SUBAPPLICATION Uebung_012d_AR (* Numeric Value Input PHYS und Speichern NVS (AR Adapter, plain) *)
  (* Standard: 61499-2; Description: Copyright (c) 2026 Meisterschulen am Ostbahnhof This program and the accompanying materials are made available under the terms of the Eclipse Public License 2.0 which is available at https://www.eclipse.org/legal/epl-2.0/ SPDX-License-Identifier: EPL-2.0 *)
  (* Version 1.0, 2026-04-24, Franz Höpfinger, Meisterschulen am Ostbahnhof, AR adapter variant of Uebung_012d, plain without subapp *)
  PACKAGE Uebungen;
  IMPORT Uebungen::const::NVS::NVS_Keys::KEY_I1_STORE;
  IMPORT Uebungen::const::UT::DefaultPool_Numeric::InputNumber_I3;
  IMPORT Uebungen::const::UT::DefaultPool_Numeric::OutputNumber_N3;
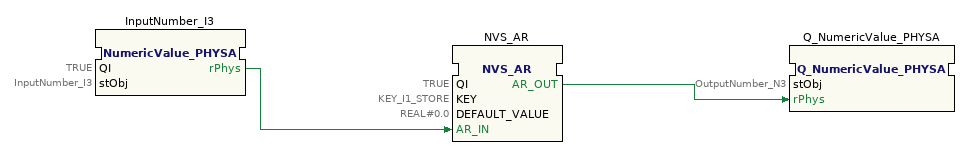
  FBS
    InputNumber_I3 : isobus::UT::io::NumericValue::NumericValue_PHYSA(QI := TRUE, stObj := InputNumber_I3);
    NVS_AR : logiBUS::storage::esp32_nvs::NVS_AR(QI := TRUE, KEY := KEY_I1_STORE, DEFAULT_VALUE := REAL#0.0);
    Q_NumericValue_PHYSA : isobus::UT::Q::Q_NumericValue_PHYSA(stObj := OutputNumber_N3);
  END_FBS
  ADAPTER_CONNECTIONS
    InputNumber_I3.rPhys TO NVS_AR.AR_IN;
    NVS_AR.AR_OUT TO Q_NumericValue_PHYSA.rPhys;
  END_CONNECTIONS
END_SUBAPPLICATION
